% RSLogix 500 project CONVEYORBELT_BAK010.RSS, saved by version 12.00.00.00 %
PROJECT "UNTITLED"    % processor: Bul.1763 MicroLogix 1100 Series B %

PROGRAM FILES
  LAD 2 "MAIN"  3 rungs
  LAD 3 "DIGITAL IO"  8 rungs
  LAD 4 "CONTROL"  12 rungs

DATA FILES
  O0 OUTPUT  4 elements
  I1 INPUT  6 elements
  S2 STATUS  66 elements
  B3 BINARY  1 elements
  T4 TIMER  3 elements
  C5 COUNTER  1 elements
  R6 CONTROL  1 elements
  N7 INTEGER  1 elements
  F8 FLOAT  1 elements

LADDER 2 "MAIN"
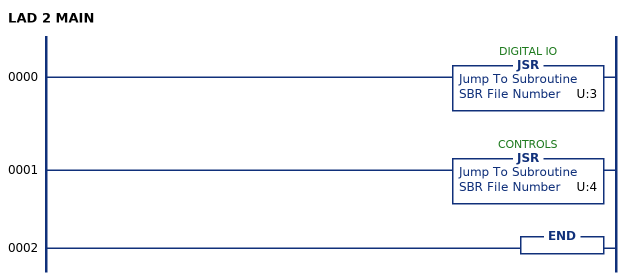
% Rung: 0 %
SOR JSR U:3 EOR
%   U:3  "DIGITAL IO" %
% Rung: 1 %
SOR JSR U:4 EOR
%   U:4  "CONTROLS" %
% Rung: 2 %
SOR END EOR

LADDER 3 "DIGITAL IO"
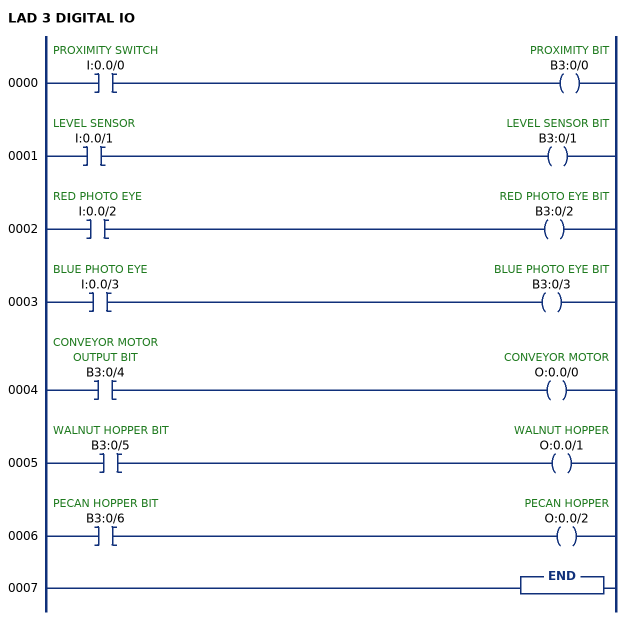
% Rung: 0 %
SOR XIC I:0.0/0 OTE B3:0/0 EOR
%   I:0.0/0  "PROXIMITY SWITCH" %
%   B3:0/0  "PROXIMITY BIT" %
% Rung: 1 %
SOR XIC I:0.0/1 OTE B3:0/1 EOR
%   I:0.0/1  "LEVEL SENSOR" %
%   B3:0/1  "LEVEL SENSOR BIT" %
% Rung: 2 %
SOR XIC I:0.0/2 OTE B3:0/2 EOR
%   I:0.0/2  "RED PHOTO EYE" %
%   B3:0/2  "RED PHOTO EYE BIT" %
% Rung: 3 %
SOR XIC I:0.0/3 OTE B3:0/3 EOR
%   I:0.0/3  "BLUE PHOTO EYE" %
%   B3:0/3  "BLUE PHOTO EYE BIT" %
% Rung: 4 %
SOR XIC B3:0/4 OTE O:0.0/0 EOR
%   B3:0/4  "CONVEYOR MOTOR OUTPUT BIT" %
%   O:0.0/0  "CONVEYOR MOTOR" %
% Rung: 5 %
SOR XIC B3:0/5 OTE O:0.0/1 EOR
%   B3:0/5  "WALNUT HOPPER BIT" %
%   O:0.0/1  "WALNUT HOPPER" %
% Rung: 6 %
SOR XIC B3:0/6 OTE O:0.0/2 EOR
%   B3:0/6  "PECAN HOPPER BIT" %
%   O:0.0/2  "PECAN HOPPER" %
% Rung: 7 %
SOR END EOR

LADDER 4 "CONTROL"
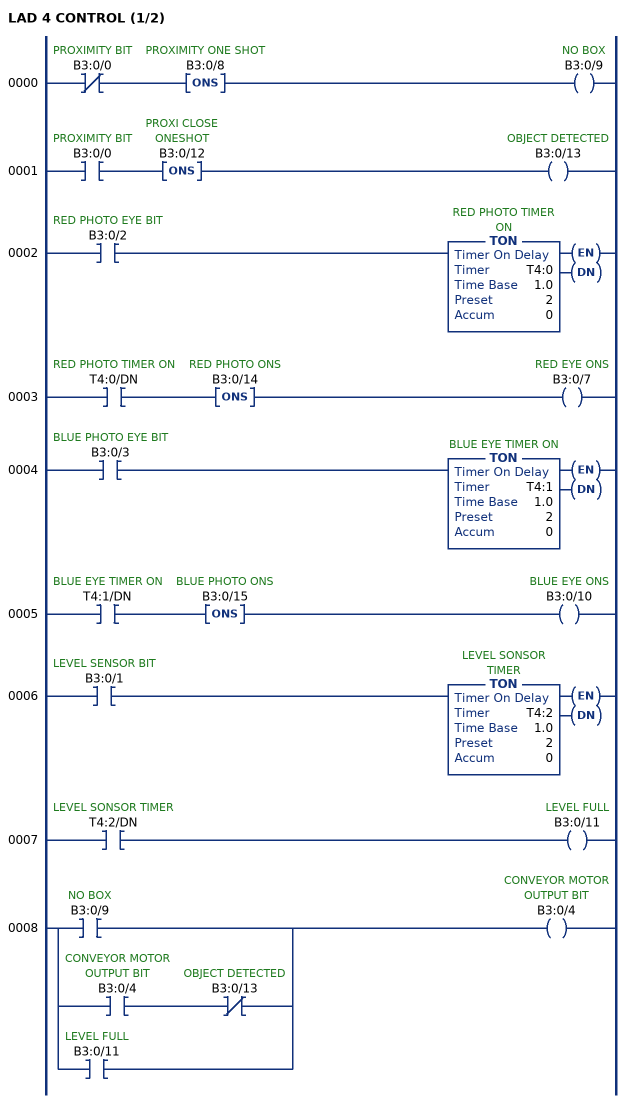
% Rung: 0 %
SOR XIO B3:0/0 ONS B3:0/8 OTE B3:0/9 EOR
%   B3:0/0  "PROXIMITY BIT" %
%   B3:0/8  "PROXIMITY ONE SHOT" %
%   B3:0/9  "NO BOX" %
% Rung: 1 %
SOR XIC B3:0/0 ONS B3:0/12 OTE B3:0/13 EOR
%   B3:0/0  "PROXIMITY BIT" %
%   B3:0/12  "PROXI CLOSE ONESHOT" %
%   B3:0/13  "OBJECT DETECTED" %
% Rung: 2 %
SOR XIC B3:0/2 TON T4:0 1.0 2 0 EOR
%   B3:0/2  "RED PHOTO EYE BIT" %
%   T4:0  "RED PHOTO TIMER ON" %
% Rung: 3 %
SOR XIC T4:0/DN ONS B3:0/14 OTE B3:0/7 EOR
%   T4:0  "RED PHOTO TIMER ON" %
%   B3:0/14  "RED PHOTO ONS" %
%   B3:0/7  "RED EYE ONS" %
% Rung: 4 %
SOR XIC B3:0/3 TON T4:1 1.0 2 0 EOR
%   B3:0/3  "BLUE PHOTO EYE BIT" %
%   T4:1  "BLUE EYE TIMER ON" %
% Rung: 5 %
SOR XIC T4:1/DN ONS B3:0/15 OTE B3:0/10 EOR
%   T4:1  "BLUE EYE TIMER ON" %
%   B3:0/15  "BLUE PHOTO ONS" %
%   B3:0/10  "BLUE EYE ONS" %
% Rung: 6 %
SOR XIC B3:0/1 TON T4:2 1.0 2 0 EOR
%   B3:0/1  "LEVEL SENSOR BIT" %
%   T4:2  "LEVEL SONSOR TIMER" %
% Rung: 7 %
SOR XIC T4:2/DN OTE B3:0/11 EOR
%   T4:2  "LEVEL SONSOR TIMER" %
%   B3:0/11  "LEVEL FULL" %
% Rung: 8 %
SOR BST XIC B3:0/9 NXB XIC B3:0/4 XIO B3:0/13 NXB XIC B3:0/11 BND OTE B3:0/4 EOR
%   B3:0/9  "NO BOX" %
%   B3:0/4  "CONVEYOR MOTOR OUTPUT BIT" %
%   B3:0/13  "OBJECT DETECTED" %
%   B3:0/11  "LEVEL FULL" %

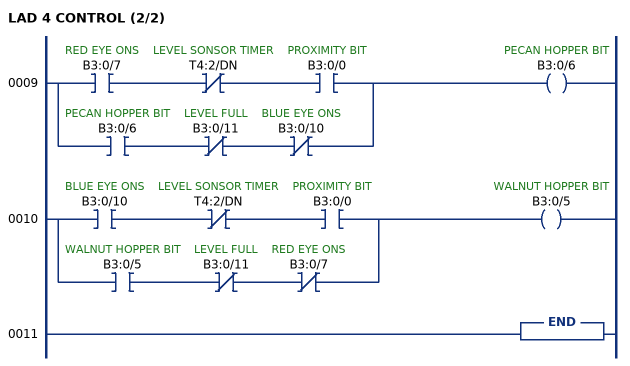
% Rung: 9 %
SOR BST XIC B3:0/7 XIO T4:2/DN XIC B3:0/0 NXB XIC B3:0/6 XIO B3:0/11 XIO B3:0/10 BND OTE B3:0/6 EOR
%   B3:0/7  "RED EYE ONS" %
%   T4:2  "LEVEL SONSOR TIMER" %
%   B3:0/0  "PROXIMITY BIT" %
%   B3:0/6  "PECAN HOPPER BIT" %
%   B3:0/11  "LEVEL FULL" %
%   B3:0/10  "BLUE EYE ONS" %
% Rung: 10 %
SOR BST XIC B3:0/10 XIO T4:2/DN XIC B3:0/0 NXB XIC B3:0/5 XIO B3:0/11 XIO B3:0/7 BND OTE B3:0/5 EOR
%   B3:0/10  "BLUE EYE ONS" %
%   T4:2  "LEVEL SONSOR TIMER" %
%   B3:0/0  "PROXIMITY BIT" %
%   B3:0/5  "WALNUT HOPPER BIT" %
%   B3:0/11  "LEVEL FULL" %
%   B3:0/7  "RED EYE ONS" %
% Rung: 11 %
SOR END EOR

OTHER DOCUMENTED ADDRESSES
  N7:0/0  "PECAN WALNUT ACIVATION MODE"

DATA TABLE (non-zero values as saved)
DATA T4
% .PRE .ACC %
% T4:0 % 2 0
% T4:1 % 2 0
% T4:2 % 2 0
